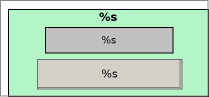
VISUALIZATION VISU_ECOMODE_EVAP  // 209x97
    RoundedRectangle (8,9 201x88), "%s", text list: 'TextList_EcoMode', text index: 8
    RoundedRectangle (45,27 128x26), "%s", colour toggle: PRG_EVAP.VISU_STOP_ECO_MANU, text list: 'TextList_EcoMode', text index: 10
    Button (37,59 145x30), "%s", text list: 'TextList_EcoMode', text index: 6
        toggle PRG_EVAP.VISU_STOP_ECO_MANU
END_VISUALIZATION

(* stored: Version 1.1.0.1, ProductVersion 3.1.4024.10
   Visu VISU_ECOMODE_EVAP: Id {c4f8f374-08db-4a36-9132-69ba62c319ca} *)
